Staubli VAL3: getLoop.pgx

public program getLoop(bool& x_bLoop[])
begin
  // get the loop status
  x_bLoop=saveCycle:bLoop
end
